TYPE LEDCommands :
STRUCT
	
	fill 		: USINT := 1;
	clear 		: USINT	:= 2;
	copy 		: USINT	:= 3;
	movePixel 	: USINT	:= 4;
	reverse 	: USINT	:= 7;
END_STRUCT
END_TYPE

(* stored: Version 1.1.0.1, ProductVersion 3.1.4026.18
   DUT LEDCommands: Id {a01da5a3-4b7e-4fb6-be4f-f38e0b7ed786} *)
